{attribute 'qualified_only'}
{attribute 'strict'}
TYPE SetPositionMode :
(
	Absolute,
	Relative
);
END_TYPE

(* stored: Version 1.1.0.1, ProductVersion 3.1.4024.12
   DUT SetPositionMode: Id {137c3cb7-ea9a-0600-1643-8418028ab866} *)
